// TwinCAT 3 PLC project Untitled1
// ProgramVersion: 3.1.4024.0
// libraries:
//   Tc2_Standard, * (Beckhoff Automation GmbH)
//   Tc2_System, * (Beckhoff Automation GmbH)
//   Tc3_Module, * (Beckhoff Automation GmbH)
// project tree:
//   DUTs/ tyMachineMode.TcDUT, tyPushButtonsControlBlock.TcDUT
//   GVLs/ GVL.TcGVL
//   / PlcTask.TcTTO
//   POUs/ MachineControlMode.TcPOU, MAIN.TcPOU
// real-time tasks:
//   TASK PlcTask: cycle T#10ms, priority 20, ADS port 350

CONFIGURATION Untitled1
    RESOURCE PLC ON TwinCAT3
        TASK PlcTask(INTERVAL := T#10ms, PRIORITY := 20);
        PROGRAM MAIN WITH PlcTask : MAIN;
    END_RESOURCE
END_CONFIGURATION

// ---- DUTs/tyMachineMode.TcDUT
TYPE tyMachineMode :
STRUCT
	MashineInRunMode :BOOL := FALSE;
	MashineInStopMode :BOOL := TRUE;
END_STRUCT
END_TYPE

// ---- DUTs/tyPushButtonsControlBlock.TcDUT
TYPE tyPushButtonsControlBlock :
STRUCT
bRunPushButton AT %I* : BOOL;
bStopPushButton	AT %I* : BOOL;
bResetPushButton	AT %I* : BOOL;
END_STRUCT
END_TYPE

// ---- GVLs/GVL.TcGVL
{attribute 'qualified_only'}
VAR_GLOBAL
	bGlobalReset : bool := false ;  
END_VAR

// ---- POUs/MAIN.TcPOU
PROGRAM MAIN
VAR
	MachineControll : MachineControlMode ; 
	
END_VAR

MachineControll();

END_PROGRAM

// ---- POUs/MachineControlMode.TcPOU
FUNCTION_BLOCK MachineControlMode
VAR_INPUT
	ControlPushButtonBlock :tyPushButtonsControlBlock;	
END_VAR
VAR_OUTPUT
END_VAR
VAR
	MachineMode :tyMachineMode;
	R_TrigRunPushBotton :R_TRIG; 
	R_TrigStopPushBotton :R_TRIG; 
END_VAR

//=============================================================================
// Dmitri Raihtsaum - Copyright 2023
// Created By: Dmitri Raihtsaum
//-----------------------------------------------------------------------------
// Tested with:   Twincat 3 
// Engineering:   Twincat 3 
// Functionality: Machine controll pushbuttons logic for training
// Date: 01.04.2023
// Rev 0.1
//=============================================================================

// Mapping 
R_TrigRunPushBotton(clk:=ControlPushButtonBlock.bRunPushButton ); 
R_TrigStopPushBotton(clk:=ControlPushButtonBlock.bStopPushButton ); 
// Protection 
IF MachineMode.MashineInRunMode AND MachineMode.MashineInStopMode THEN
	MachineMode.MashineInRunMode  := FALSE; 
	MachineMode.MashineInStopMode := TRUE; 
END_IF;
IF NOT MachineMode.MashineInRunMode AND NOT  MachineMode.MashineInStopMode THEN
	MachineMode.MashineInRunMode  := FALSE; 
	MachineMode.MashineInStopMode := TRUE; 
END_IF;
// Logic 
IF R_TrigStopPushBotton.Q THEN 
	MachineMode.MashineInRunMode  := FALSE; 
	MachineMode.MashineInStopMode := TRUE  ; 
END_IF
IF R_TrigRunPushBotton.Q THEN 
	MachineMode.MashineInRunMode  := TRUE; 
	MachineMode.MashineInStopMode := FALSE ; 
END_IF
//Global Reset 
IF MachineMode.MashineInStopMode AND ControlPushButtonBlock.bResetPushButton THEN 
	GVL.bGlobalReset := TRUE;
	ELSE 
		GVL.bGlobalReset := FALSE;
END_IF;

///////////////////////END///////////////////////

END_FUNCTION_BLOCK
